FUNCTION ck_real_value :ck_real_flag_data
//return ck_real_flag_data struct
VAR_INPUT
	//imput Vision_data struct 
	data: Vision_data;
END_VAR
VAR
END_VAR


//check if two of tree values are the same, to avoid bad variables intercahnages between vision system and plc
//return flag ck_real_flag_data[0] to indicate is correct, and one real value ck_real_value[1] 
IF data.Val2=data.Val3 THEN
	ck_real_value.Flag:=TRUE;
	ck_real_value.Value:=data.Val2;
ELSIF data.Val1=data.Val3 THEN
	ck_real_value.Flag:=TRUE;
	ck_real_value.Value:=data.Val3;
ELSIF data.Val1=data.Val2 THEN
	ck_real_value.Flag:=TRUE;
	ck_real_value.Value:=data.Val2;
ELSIF (data.Val1=data.Val2 AND data.Val1=data.Val3 AND data.Val2=data.Val3) THEN	
	ck_real_value.Flag:=TRUE;
	ck_real_value.Value:=data.Val1;
ELSE	
	ck_real_value.Flag:=FALSE;
END_IF

END_FUNCTION

(* stored: Version 1.1.0.1, ProductVersion 3.1.4024.4
   POU ck_real_value: Id {78e4faa4-d0aa-4612-956f-b10eebb1f419}, SpecialFunc None *)
